PROGRAM MAIN
VAR
	GetTime: NT_GetTime;

	getLocalAMS: FB_GetLocalAmsNetId;
	

	oneSec: fb_flasher;
	tenSec: fb_flasher;
	
	oneMSec: fb_flasher;
END_VAR
VAR // added by the converter: edge detectors and wires of the graphical bodies
    _rt1, _rt2 : R_TRIG;
    _w1, _w2 : BOOL;
END_VAR

//call PLC data
actPLC();

//call init data for machine
actInit();

//call clock memory
actClockMemory();

//call all diagnostics
actDiag();

//call base machine

//call HMI
//calls logic to drive the HMI
pouHMI();

//call machine base
pouMachine();

//call station 1
//calls motions only associated with station 1
pouStation1();

//call station 2
pouStation2();

//call station 3
pouStation3();

//call station 4
pouStation4();

//call station 5
pouStation5();

//call station 6
pouStation6();

//there are only ever 6 maximum stations

ACTION actClockMemory:
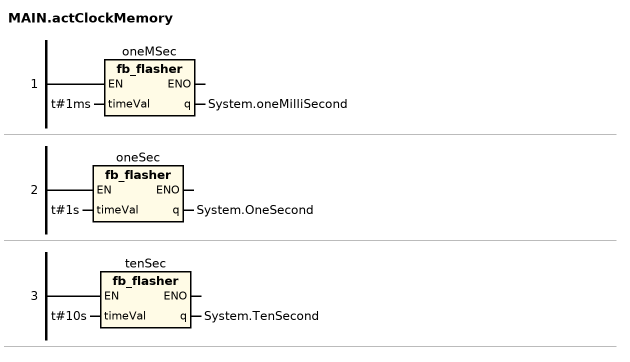
// NETWORK 1
oneMSec(timeVal := t#1ms, q => System.oneMilliSecond); // fb_flasher

// NETWORK 2
oneSec(timeVal := t#1s, q => System.OneSecond); // fb_flasher

// NETWORK 3
tenSec(timeVal := t#10s, q => System.TenSecond); // fb_flasher
END_ACTION

ACTION actDiag:
//call diag blocks
pouDPDiag();
pouEtherCATdiag();
pouPROFINETdiag();
END_ACTION

ACTION actInit:
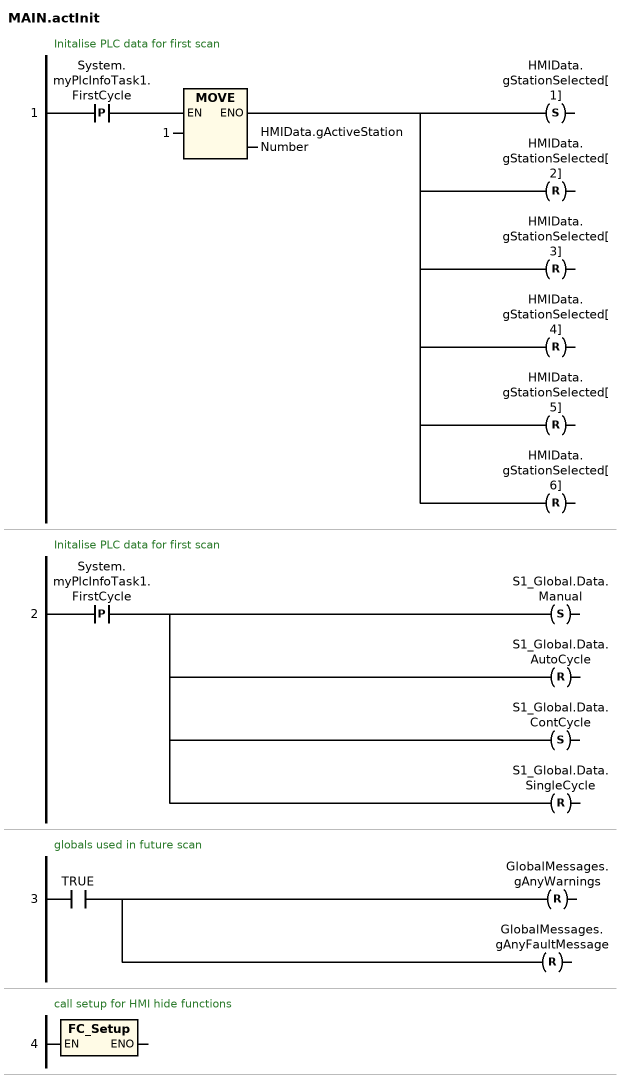
// NETWORK 1
// Initalise PLC data for first scan
_rt1(CLK := System.myPlcInfoTask1.FirstCycle);
_w1 := _rt1.Q;
IF _w1 THEN HMIData.gActiveStationNumber := 1; END_IF
HMIData.gStationSelected[1] S= _w1;
HMIData.gStationSelected[2] R= _w1;
HMIData.gStationSelected[3] R= _w1;
HMIData.gStationSelected[4] R= _w1;
HMIData.gStationSelected[5] R= _w1;
HMIData.gStationSelected[6] R= _w1;

// NETWORK 2
// Initalise PLC data for first scan
_rt2(CLK := System.myPlcInfoTask1.FirstCycle);
S1_Global.Data.Manual S= _rt2.Q;
S1_Global.Data.AutoCycle R= _rt2.Q;
S1_Global.Data.ContCycle S= _rt2.Q;
S1_Global.Data.SingleCycle R= _rt2.Q;

// NETWORK 3
// globals used in future scan
GlobalMessages.gAnyWarnings R= TRUE;
GlobalMessages.gAnyFaultMessage R= TRUE;

// NETWORK 4
// call setup for HMI hide functions
FC_Setup();
END_ACTION

ACTION actPLC:
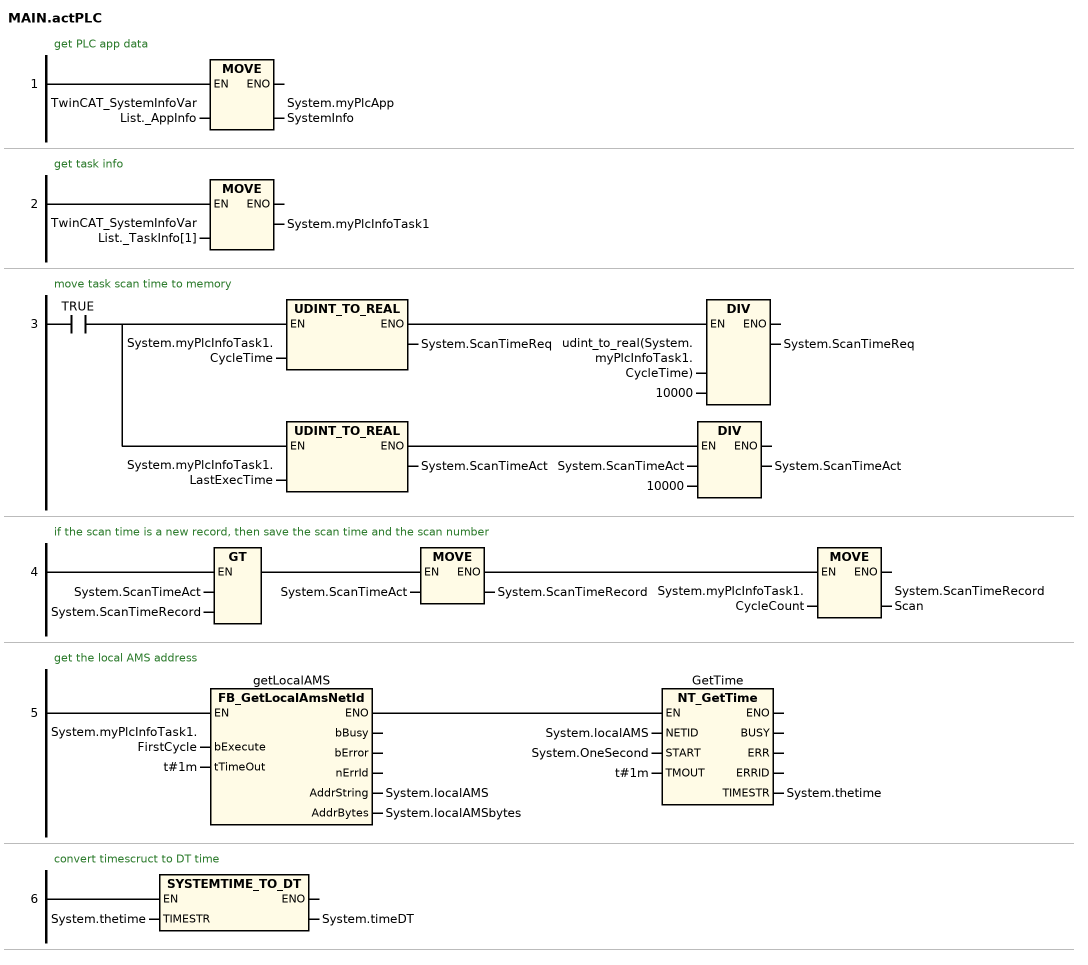
// NETWORK 1
// get PLC app data
System.myPlcAppSystemInfo := TwinCAT_SystemInfoVarList._AppInfo;

// NETWORK 2
// get task info
System.myPlcInfoTask1 := TwinCAT_SystemInfoVarList._TaskInfo[1];

// NETWORK 3
// move task scan time to memory
System.ScanTimeReq := UDINT_TO_REAL(System.myPlcInfoTask1.CycleTime);
System.ScanTimeReq := (udint_to_real(System.myPlcInfoTask1.CycleTime)) / 10000;
System.ScanTimeAct := UDINT_TO_REAL(System.myPlcInfoTask1.LastExecTime);
System.ScanTimeAct := System.ScanTimeAct / 10000;

// NETWORK 4
// if the scan time is a new record, then save the scan time and the scan number
_w2 := System.ScanTimeAct > System.ScanTimeRecord;
IF _w2 THEN System.ScanTimeRecord := System.ScanTimeAct; END_IF
IF _w2 THEN System.ScanTimeRecordScan := System.myPlcInfoTask1.CycleCount; END_IF

// NETWORK 5
// get the local AMS address
getLocalAMS(
    bExecute := System.myPlcInfoTask1.FirstCycle,
    tTimeOut := t#1m,
    AddrString => System.localAMS,
    AddrBytes => System.localAMSbytes); // FB_GetLocalAmsNetId
GetTime(NETID := System.localAMS, START := System.OneSecond, TMOUT := t#1m, TIMESTR => System.thetime); // NT_GetTime

// NETWORK 6
// convert timescruct to DT time
System.timeDT := SYSTEMTIME_TO_DT(TIMESTR := System.thetime);
END_ACTION

END_PROGRAM

(* stored: Version 1.1.0.1, ProductVersion 3.1.4024.12
   POU MAIN: Id {71925003-04a7-4f4b-805b-2cb8426e0ca0}, SpecialFunc None
   Action actClockMemory: Id {ada9ce1e-1cab-4114-94fc-89c6fb0a28ae}
   Action actDiag: Id {64b32e1c-14ce-4e5e-ba1b-93c63e0d0e72}
   Action actInit: Id {647dce60-d775-41b1-a8f3-8b905b314130}
   Action actPLC: Id {19d58927-e0ae-4a22-9363-412c9c6d376e} *)
